{attribute 'GeneratedUsingTerminal: EP4174-0002-0016'}
{attribute addProperty BoxType "EP4174-0002-0016"}
{attribute addProperty Id "Analog_outputAT %Q*INT2"}
{attribute addProperty CRC "3128867708"}
{attribute addProperty Size "2"}
TYPE AO_Output_Channel_BA7EBB7C EXTENDS OutputBase_10CEE7DE :
STRUCT
	{attribute addProperty Name "Analog_output"}
	Analog_output AT %Q* : INT;
END_STRUCT
END_TYPE

(* stored: Version 1.2.0.0, ProductVersion 3.1.4024.11
   DUT AO_Output_Channel_BA7EBB7C: Id {5a2caabb-6219-4784-b8fc-71405f279efc} *)
